// TIA Portal V20 export
TYPE "UDT_PathCmd"
TITLE = Buffered-path command element (V4.0 palletizing)
// One command in the buffered-path command list (GDB_PalletizingPath.aCmd). Authored by FB_AutoCtrl_Palletizing REGION 1, executed by REGION 4.
   STRUCT
      i16_CmdType : Int;   // Command type: 0 = END_OF_PATH, 1 = MOVE, 2 = GRIPPER, 3 = WAIT_ARRIVAL
      x : LReal;   // MOVE: target Cartesian X [mm]
      y : LReal;   // MOVE: target Cartesian Y [mm]
      z : LReal;   // MOVE: target Cartesian Z [mm]
      "a" : LReal;   // MOVE: target wrist orientation A [deg]
      lr_Velocity : LReal;   // MOVE: path velocity [mm/s]
      i16_BufferMode : Int;   // MOVE: MC_MoveLinearAbsolute BufferMode for this command -- 1 = stop at this point (BM_BUFFERED), 5 = blend through it (BM_BLENDING_HIGH). Never 0 (MC_Aborting is invalid for a kinematic path -> 16#80B2).
      lr_DwellMs : LReal;   // GRIPPER: grip/release settle hold time [ms]
      bo_GripperGrip : Bool;   // GRIPPER: level value written to GDB_Control.bo_gripperGrip
      bo_GripperRelease : Bool;   // GRIPPER: if TRUE, pulse GDB_Control.bo_gripperRelease for the dwell then drop it
      bo_IsBoxEnd : Bool;   // MOVE: TRUE on the PLACE_RETRACT move that completes a box -- increments statBoxesPlaced and re-arms the spawn request
      i16_HmiStep : Int;   // Value published to GDB_PalletizingCmd.i16_PalletStep when this command becomes active -- preserves the HMI 1..48 step display
   END_STRUCT;
END_TYPE
